FUNCTION_BLOCK FB_DescargarPieza_SFC

VAR_IN_OUT
	    TpoPinza: TIME;
END_VAR

VAR_INPUT
    // SFC-Flags
    SFCPause: BOOL;
    SFCReset: BOOL;
    
    // Indicadores de sincronizacion
    Ack: BOOL := TRUE;
    Execute: BOOL;
    
    // Entradas
    DescargadorDetras : BOOL;
	DescargadorDelante : BOOL;
	DescargadorArriba : BOOL;
	DescargadorAbajo : BOOL;
END_VAR
VAR_OUTPUT
    // Indicadores de sincronizacion
    Done: BOOL;
    Ready: BOOL;
    
    // Salidas
    DescargadorAvanza AT %Q*: BOOL;
	DescargadorBaja AT %Q*: BOOL;
	DescargadorCierra AT %Q*: BOOL;
END_VAR
VAR
END_VAR

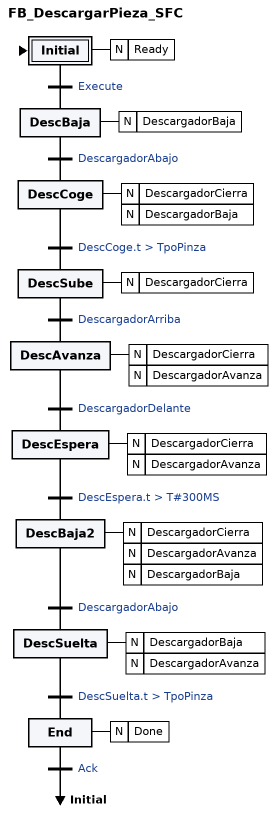
INITIAL_STEP Initial:
    Ready(N);
END_STEP
TRANSITION FROM Initial TO DescBaja
    := Execute;
END_TRANSITION
STEP DescBaja:
    DescargadorBaja(N);
END_STEP
TRANSITION FROM DescBaja TO DescCoge
    := DescargadorAbajo;
END_TRANSITION
STEP DescCoge:
    DescargadorCierra(N);
    DescargadorBaja(N);
END_STEP
TRANSITION FROM DescCoge TO DescSube
    := DescCoge.t > TpoPinza;
END_TRANSITION
STEP DescSube:
    DescargadorCierra(N);
END_STEP
TRANSITION FROM DescSube TO DescAvanza
    := DescargadorArriba;
END_TRANSITION
STEP DescAvanza:
    DescargadorCierra(N);
    DescargadorAvanza(N);
END_STEP
TRANSITION FROM DescAvanza TO DescEspera
    := DescargadorDelante;
END_TRANSITION
STEP DescEspera:
    DescargadorCierra(N);
    DescargadorAvanza(N);
END_STEP
TRANSITION FROM DescEspera TO DescBaja2
    := DescEspera.t > T#300MS;
END_TRANSITION
STEP DescBaja2:
    DescargadorCierra(N);
    DescargadorAvanza(N);
    DescargadorBaja(N);
END_STEP
TRANSITION FROM DescBaja2 TO DescSuelta
    := DescargadorAbajo;
END_TRANSITION
STEP DescSuelta:
    DescargadorBaja(N);
    DescargadorAvanza(N);
END_STEP
TRANSITION FROM DescSuelta TO End
    := DescSuelta.t > TpoPinza;
END_TRANSITION
STEP End:
    Done(N);
END_STEP
TRANSITION FROM End TO Initial
    := Ack;
END_TRANSITION

END_FUNCTION_BLOCK

(* stored: Version 1.1.0.1, ProductVersion 3.1.4024.9
   POU FB_DescargarPieza_SFC: Id {1f015f68-c158-45c4-9c66-eb9f2726e884}, SpecialFunc None *)
